PROGRAM MAIN
VAR
    Initialize	:	BOOL := TRUE;

    fbLogHandler : FB_LogHandler;
    fbEcatDiag : FB_EcatDiagWrapper;

    {attribute 'pytmc' := '
        pv: Arbiter:Link:HGVPU
        link: USEG:UNDH:
    '}
    fbHgvpu : FB_Hgvpu;

    {attribute 'pytmc' := '
        pv: Arbiter:Link:SXU
        link: USEG:UNDS:
    '}
    fbSxu : FB_SXU;

END_VAR

//Arbiter PLC

IF Initialize THEN
    Initialize := FALSE;
END_IF

// Ethercat Diagnostics
fbEcatDiag();

///////////////////////////////////////////////////
// This code should be disabled or removed in deployment
// Might have a switch to change to simulation mode
MachineSimulation();
Testing();
///////////////////////////////////////////////////

//Update current BP
CurrentBPUpdate();

// PMPS Functionality
PMPS_Arbiter();


fbLogHandler();

ACTION Initialize:

END_ACTION

END_PROGRAM

(* stored: Version 1.1.0.1, ProductVersion 3.1.4022.18
   POU MAIN: Id {8a7bcfd2-1a2b-4363-aa47-c19391bf1f9c}, SpecialFunc None
   Action Initialize: Id {b0ee480a-3d4b-001d-04c4-43cdc47895c8} *)
